# B&R Automation Studio project PT_KB_V01 (part 10)

#### Cyclic.st - Cyclic code
```iecst
PROGRAM _CYCLIC
	(* ======================================================================== *)
	(* 1) Komunikacioni, pogonski i AirRelease izvori                           *)
	(* ======================================================================== *)
	PT_Alarm.Comm.BRB2.Active := PGRad_Cmd.Aktivan AND NOT PGRad_BRB2Watchdog.Valid;
	PT_Alarm.Comm.IEBKB1.Active := PGRad_Cmd.Aktivan
		AND (PGRad.Ctrl.SelektovaniIzvor = _02_IEBKB1)
		AND (NOT PGRad_IEBKB1Prepared.CommValid OR NOT PGRad_IEBKB1Prepared.HeartbeatValid);
	PT_Alarm.Comm.BRB2RemoteFault.Active := PGRad_BRB2.BRB2Fault;
	PT_Alarm.Drive.PG_Pu01_VFD.Active := PG.Act.Pu._1.Alarm_FR;
	PT_Alarm.Drive.PG_Pu01_CAN.Active := PG.Act.Pu._1.Alarm_CAN;
	PT_Alarm.Drive.PG_Pu02_VFD.Active := PG.Act.Pu._2.Alarm_FR;
	PT_Alarm.Drive.PG_Pu02_CAN.Active := PG.Act.Pu._2.Alarm_CAN;
	PT_Alarm.AirRelease.PG_PV03.Active := PGRad_AirRelease.PV03.FB.AR_Output.AlarmActive;
	PT_Alarm.AirRelease.PG_PV04.Active := PGRad_AirRelease.PV04.FB.AR_Output.AlarmActive;

	PT_Alarm.Comm.BRB2.ResetAllowed := NOT PT_Alarm.Comm.BRB2.Active;
	PT_Alarm.Comm.IEBKB1.ResetAllowed := NOT PT_Alarm.Comm.IEBKB1.Active;
	PT_Alarm.Comm.BRB2RemoteFault.ResetAllowed := NOT PT_Alarm.Comm.BRB2RemoteFault.Active;
	PT_Alarm.Drive.PG_Pu01_VFD.ResetAllowed := NOT PT_Alarm.Drive.PG_Pu01_VFD.Active;
	PT_Alarm.Drive.PG_Pu01_CAN.ResetAllowed := NOT PT_Alarm.Drive.PG_Pu01_CAN.Active;
	PT_Alarm.Drive.PG_Pu02_VFD.ResetAllowed := NOT PT_Alarm.Drive.PG_Pu02_VFD.Active;
	PT_Alarm.Drive.PG_Pu02_CAN.ResetAllowed := NOT PT_Alarm.Drive.PG_Pu02_CAN.Active;
	PT_Alarm.AirRelease.PG_PV03.ResetAllowed := PGRad_AirRelease.PV03.FB.AR_Output.ResetAllowed;
	PT_Alarm.AirRelease.PG_PV04.ResetAllowed := PGRad_AirRelease.PV04.FB.AR_Output.ResetAllowed;
	PT_Alarm.AirRelease.PG_PV03.SourceCode := PGRad_AirRelease.PV03.FB.AR_Output.FaultCode;
	PT_Alarm.AirRelease.PG_PV04.SourceCode := PGRad_AirRelease.PV04.FB.AR_Output.FaultCode;

	(* ======================================================================== *)
	(* 2) IO_Modules: status, latch, potvrda i STOP svih fizickih modula       *)
	(* ======================================================================== *)
	PT_Alarm.IO.X20AI4622.Fault := NOT PT_Alarm.IO.X20AI4622.ModuleOk;
	PT_Alarm.IO.X20AI4622a.Fault := NOT PT_Alarm.IO.X20AI4622a.ModuleOk;
	PT_Alarm.IO.X20AI4622b.Fault := NOT PT_Alarm.IO.X20AI4622b.ModuleOk;
	PT_Alarm.IO.X20AI4622c.Fault := NOT PT_Alarm.IO.X20AI4622c.ModuleOk;
	PT_Alarm.IO.X20AI4622d.Fault := NOT PT_Alarm.IO.X20AI4622d.ModuleOk;
	PT_Alarm.IO.X20AO4622.Fault := NOT PT_Alarm.IO.X20AO4622.ModuleOk;
	PT_Alarm.IO.X20AO4622a.Fault := NOT PT_Alarm.IO.X20AO4622a.ModuleOk;
	PT_Alarm.IO.X20AO4622b.Fault := NOT PT_Alarm.IO.X20AO4622b.ModuleOk;
	PT_Alarm.IO.X20DI9371.Fault := NOT PT_Alarm.IO.X20DI9371.ModuleOk;
	PT_Alarm.IO.X20DI9371a.Fault := NOT PT_Alarm.IO.X20DI9371a.ModuleOk;
	PT_Alarm.IO.X20DI9371b.Fault := NOT PT_Alarm.IO.X20DI9371b.ModuleOk;
	PT_Alarm.IO.X20DO9322.Fault := NOT PT_Alarm.IO.X20DO9322.ModuleOk;
	PT_Alarm.IO.X20DO9322a.Fault := NOT PT_Alarm.IO.X20DO9322a.ModuleOk;
	PT_Alarm.IO.X20BC0083.Fault := NOT PT_Alarm.IO.X20BC0083.ModuleOk;
	PT_Alarm.IO.X20PS9400.Fault := NOT PT_Alarm.IO.X20PS9400.ModuleOk;
	PT_Alarm.IO.X20BT9100a.Fault := NOT PT_Alarm.IO.X20BT9100a.ModuleOk;
	PT_Alarm.IO.X67AI1323.Fault := NOT PT_Alarm.IO.X67AI1323.ModuleOk;
	PT_Alarm.IO.X67AI1333b.Fault := NOT PT_Alarm.IO.X67AI1333b.ModuleOk;
	PT_Alarm.IO.X67DI1371_L12.Fault := NOT PT_Alarm.IO.X67DI1371_L12.ModuleOk;
	PT_Alarm.IO.X67DM1321_L12.Fault := NOT PT_Alarm.IO.X67DM1321_L12.ModuleOk;
	PT_Alarm.IO.X20AI4622.Code := 41001; PT_Alarm.IO.X20AI4622.ResetAllowed := NOT PT_Alarm.IO.X20AI4622.Fault; PT_Alarm.IO.X20AI4622.Blocking := TRUE;
	PT_Alarm.IO.X20AI4622a.Code := 41002; PT_Alarm.IO.X20AI4622a.ResetAllowed := NOT PT_Alarm.IO.X20AI4622a.Fault; PT_Alarm.IO.X20AI4622a.Blocking := TRUE;
	PT_Alarm.IO.X20AI4622b.Code := 41003; PT_Alarm.IO.X20AI4622b.ResetAllowed := NOT PT_Alarm.IO.X20AI4622b.Fault; PT_Alarm.IO.X20AI4622b.Blocking := TRUE;
	PT_Alarm.IO.X20AI4622c.Code := 41004; PT_Alarm.IO.X20AI4622c.ResetAllowed := NOT PT_Alarm.IO.X20AI4622c.Fault; PT_Alarm.IO.X20AI4622c.Blocking := TRUE;
	PT_Alarm.IO.X20AI4622d.Code := 41005; PT_Alarm.IO.X20AI4622d.ResetAllowed := NOT PT_Alarm.IO.X20AI4622d.Fault; PT_Alarm.IO.X20AI4622d.Blocking := TRUE;
	PT_Alarm.IO.X20AO4622.Code := 41101; PT_Alarm.IO.X20AO4622.ResetAllowed := NOT PT_Alarm.IO.X20AO4622.Fault; PT_Alarm.IO.X20AO4622.Blocking := TRUE;
	PT_Alarm.IO.X20AO4622a.Code := 41102; PT_Alarm.IO.X20AO4622a.ResetAllowed := NOT PT_Alarm.IO.X20AO4622a.Fault; PT_Alarm.IO.X20AO4622a.Blocking := TRUE;
	PT_Alarm.IO.X20AO4622b.Code := 41103; PT_Alarm.IO.X20AO4622b.ResetAllowed := NOT PT_Alarm.IO.X20AO4622b.Fault; PT_Alarm.IO.X20AO4622b.Blocking := TRUE;
	PT_Alarm.IO.X20DI9371.Code := 41201; PT_Alarm.IO.X20DI9371.ResetAllowed := NOT PT_Alarm.IO.X20DI9371.Fault; PT_Alarm.IO.X20DI9371.Blocking := TRUE;
	PT_Alarm.IO.X20DI9371a.Code := 41202; PT_Alarm.IO.X20DI9371a.ResetAllowed := NOT PT_Alarm.IO.X20DI9371a.Fault; PT_Alarm.IO.X20DI9371a.Blocking := TRUE;
	PT_Alarm.IO.X20DI9371b.Code := 41203; PT_Alarm.IO.X20DI9371b.ResetAllowed := NOT PT_Alarm.IO.X20DI9371b.Fault; PT_Alarm.IO.X20DI9371b.Blocking := TRUE;
	PT_Alarm.IO.X20DO9322.Code := 41301; PT_Alarm.IO.X20DO9322.ResetAllowed := NOT PT_Alarm.IO.X20DO9322.Fault; PT_Alarm.IO.X20DO9322.Blocking := TRUE;
	PT_Alarm.IO.X20DO9322a.Code := 41302; PT_Alarm.IO.X20DO9322a.ResetAllowed := NOT PT_Alarm.IO.X20DO9322a.Fault; PT_Alarm.IO.X20DO9322a.Blocking := TRUE;
	PT_Alarm.IO.X20BC0083.Code := 41401; PT_Alarm.IO.X20BC0083.ResetAllowed := NOT PT_Alarm.IO.X20BC0083.Fault; PT_Alarm.IO.X20BC0083.Blocking := TRUE;
	PT_Alarm.IO.X20PS9400.Code := 41402; PT_Alarm.IO.X20PS9400.ResetAllowed := NOT PT_Alarm.IO.X20PS9400.Fault; PT_Alarm.IO.X20PS9400.Blocking := TRUE;
	PT_Alarm.IO.X20BT9100a.Code := 41403; PT_Alarm.IO.X20BT9100a.ResetAllowed := NOT PT_Alarm.IO.X20BT9100a.Fault; PT_Alarm.IO.X20BT9100a.Blocking := TRUE;
	PT_Alarm.IO.X67AI1323.Code := 41501; PT_Alarm.IO.X67AI1323.ResetAllowed := NOT PT_Alarm.IO.X67AI1323.Fault; PT_Alarm.IO.X67AI1323.Blocking := TRUE;
	PT_Alarm.IO.X67AI1333b.Code := 41502; PT_Alarm.IO.X67AI1333b.ResetAllowed := NOT PT_Alarm.IO.X67AI1333b.Fault; PT_Alarm.IO.X67AI1333b.Blocking := TRUE;
	PT_Alarm.IO.X67DI1371_L12.Code := 41601; PT_Alarm.IO.X67DI1371_L12.ResetAllowed := NOT PT_Alarm.IO.X67DI1371_L12.Fault; PT_Alarm.IO.X67DI1371_L12.Blocking := TRUE;
	PT_Alarm.IO.X67DM1321_L12.Code := 41701; PT_Alarm.IO.X67DM1321_L12.ResetAllowed := NOT PT_Alarm.IO.X67DM1321_L12.Fault; PT_Alarm.IO.X67DM1321_L12.Blocking := TRUE;
	IF PT_Alarm.IO.X20AI4622.Fault OR PT_Alarm.IO.X20AI4622a.Fault OR PT_Alarm.IO.X20AI4622b.Fault OR PT_Alarm.IO.X20AI4622c.Fault OR PT_Alarm.IO.X20AI4622d.Fault OR PT_Alarm.IO.X20AO4622.Fault OR PT_Alarm.IO.X20AO4622a.Fault OR PT_Alarm.IO.X20AO4622b.Fault OR PT_Alarm.IO.X20DI9371.Fault OR PT_Alarm.IO.X20DI9371a.Fault OR PT_Alarm.IO.X20DI9371b.Fault OR PT_Alarm.IO.X20DO9322.Fault OR PT_Alarm.IO.X20DO9322a.Fault OR PT_Alarm.IO.X20BC0083.Fault OR PT_Alarm.IO.X20PS9400.Fault OR PT_Alarm.IO.X20BT9100a.Fault OR PT_Alarm.IO.X67AI1323.Fault OR PT_Alarm.IO.X67AI1333b.Fault OR PT_Alarm.IO.X67DI1371_L12.Fault OR PT_Alarm.IO.X67DM1321_L12.Fault THEN
		PT_Alarm.IO.X20AI4622.Latched := PT_Alarm.IO.X20AI4622.Latched OR PT_Alarm.IO.X20AI4622.Fault;
		PT_Alarm.IO.X20AI4622a.Latched := PT_Alarm.IO.X20AI4622a.Latched OR PT_Alarm.IO.X20AI4622a.Fault;
		PT_Alarm.IO.X20AI4622b.Latched := PT_Alarm.IO.X20AI4622b.Latched OR PT_Alarm.IO.X20AI4622b.Fault;
		PT_Alarm.IO.X20AI4622c.Latched := PT_Alarm.IO.X20AI4622c.Latched OR PT_Alarm.IO.X20AI4622c.Fault;
		PT_Alarm.IO.X20AI4622d.Latched := PT_Alarm.IO.X20AI4622d.Latched OR PT_Alarm.IO.X20AI4622d.Fault;
		PT_Alarm.IO.X20AO4622.Latched := PT_Alarm.IO.X20AO4622.Latched OR PT_Alarm.IO.X20AO4622.Fault;
		PT_Alarm.IO.X20AO4622a.Latched := PT_Alarm.IO.X20AO4622a.Latched OR PT_Alarm.IO.X20AO4622a.Fault;
		PT_Alarm.IO.X20AO4622b.Latched := PT_Alarm.IO.X20AO4622b.Latched OR PT_Alarm.IO.X20AO4622b.Fault;
		PT_Alarm.IO.X20DI9371.Latched := PT_Alarm.IO.X20DI9371.Latched OR PT_Alarm.IO.X20DI9371.Fault;
		PT_Alarm.IO.X20DI9371a.Latched := PT_Alarm.IO.X20DI9371a.Latched OR PT_Alarm.IO.X20DI9371a.Fault;
		PT_Alarm.IO.X20DI9371b.Latched := PT_Alarm.IO.X20DI9371b.Latched OR PT_Alarm.IO.X20DI9371b.Fault;
		PT_Alarm.IO.X20DO9322.Latched := PT_Alarm.IO.X20DO9322.Latched OR PT_Alarm.IO.X20DO9322.Fault;
		PT_Alarm.IO.X20DO9322a.Latched := PT_Alarm.IO.X20DO9322a.Latched OR PT_Alarm.IO.X20DO9322a.Fault;
		PT_Alarm.IO.X20BC0083.Latched := PT_Alarm.IO.X20BC0083.Latched OR PT_Alarm.IO.X20BC0083.Fault;
		PT_Alarm.IO.X20PS9400.Latched := PT_Alarm.IO.X20PS9400.Latched OR PT_Alarm.IO.X20PS9400.Fault;
		PT_Alarm.IO.X20BT9100a.Latched := PT_Alarm.IO.X20BT9100a.Latched OR PT_Alarm.IO.X20BT9100a.Fault;
		PT_Alarm.IO.X67AI1323.Latched := PT_Alarm.IO.X67AI1323.Latched OR PT_Alarm.IO.X67AI1323.Fault;
		PT_Alarm.IO.X67AI1333b.Latched := PT_Alarm.IO.X67AI1333b.Latched OR PT_Alarm.IO.X67AI1333b.Fault;
		PT_Alarm.IO.X67DI1371_L12.Latched := PT_Alarm.IO.X67DI1371_L12.Latched OR PT_Alarm.IO.X67DI1371_L12.Fault;
		PT_Alarm.IO.X67DM1321_L12.Latched := PT_Alarm.IO.X67DM1321_L12.Latched OR PT_Alarm.IO.X67DM1321_L12.Fault;
	END_IF;
	IF PT_Alarm.Cmd.ResetAlarmRecords THEN
		IF PT_Alarm.IO.X20AI4622.ResetAllowed THEN PT_Alarm.IO.X20AI4622.Latched := FALSE; END_IF;
		IF PT_Alarm.IO.X20AI4622a.ResetAllowed THEN PT_Alarm.IO.X20AI4622a.Latched := FALSE; END_IF;
		IF PT_Alarm.IO.X20AI4622b.ResetAllowed THEN PT_Alarm.IO.X20AI4622b.Latched := FALSE; END_IF;
		IF PT_Alarm.IO.X20AI4622c.ResetAllowed THEN PT_Alarm.IO.X20AI4622c.Latched := FALSE; END_IF;
		IF PT_Alarm.IO.X20AI4622d.ResetAllowed THEN PT_Alarm.IO.X20AI4622d.Latched := FALSE; END_IF;
		IF PT_Alarm.IO.X20AO4622.ResetAllowed THEN PT_Alarm.IO.X20AO4622.Latched := FALSE; END_IF;
		IF PT_Alarm.IO.X20AO4622a.ResetAllowed THEN PT_Alarm.IO.X20AO4622a.Latched := FALSE; END_IF;
		IF PT_Alarm.IO.X20AO4622b.ResetAllowed THEN PT_Alarm.IO.X20AO4622b.Latched := FALSE; END_IF;
		IF PT_Alarm.IO.X20DI9371.ResetAllowed THEN PT_Alarm.IO.X20DI9371.Latched := FALSE; END_IF;
		IF PT_Alarm.IO.X20DI9371a.ResetAllowed THEN PT_Alarm.IO.X20DI9371a.Latched := FALSE; END_IF;
		IF PT_Alarm.IO.X20DI9371b.ResetAllowed THEN PT_Alarm.IO.X20DI9371b.Latched := FALSE; END_IF;
		IF PT_Alarm.IO.X20DO9322.ResetAllowed THEN PT_Alarm.IO.X20DO9322.Latched := FALSE; END_IF;
		IF PT_Alarm.IO.X20DO9322a.ResetAllowed THEN PT_Alarm.IO.X20DO9322a.Latched := FALSE; END_IF;
		IF PT_Alarm.IO.X20BC0083.ResetAllowed THEN PT_Alarm.IO.X20BC0083.Latched := FALSE; END_IF;
		IF PT_Alarm.IO.X20PS9400.ResetAllowed THEN PT_Alarm.IO.X20PS9400.Latched := FALSE; END_IF;
		IF PT_Alarm.IO.X20BT9100a.ResetAllowed THEN PT_Alarm.IO.X20BT9100a.Latched := FALSE; END_IF;
		IF PT_Alarm.IO.X67AI1323.ResetAllowed THEN PT_Alarm.IO.X67AI1323.Latched := FALSE; END_IF;
		IF PT_Alarm.IO.X67AI1333b.ResetAllowed THEN PT_Alarm.IO.X67AI1333b.Latched := FALSE; END_IF;
		IF PT_Alarm.IO.X67DI1371_L12.ResetAllowed THEN PT_Alarm.IO.X67DI1371_L12.Latched := FALSE; END_IF;
		IF PT_Alarm.IO.X67DM1321_L12.ResetAllowed THEN PT_Alarm.IO.X67DM1321_L12.Latched := FALSE; END_IF;
	END_IF;
	PT_Alarm.IO.AnyFault :=
		PT_Alarm.IO.X20AI4622.Fault OR PT_Alarm.IO.X20AI4622a.Fault OR PT_Alarm.IO.X20AI4622b.Fault OR
		PT_Alarm.IO.X20AI4622c.Fault OR PT_Alarm.IO.X20AI4622d.Fault OR PT_Alarm.IO.X20AO4622.Fault OR
		PT_Alarm.IO.X20AO4622a.Fault OR PT_Alarm.IO.X20AO4622b.Fault OR PT_Alarm.IO.X20DI9371.Fault OR
		PT_Alarm.IO.X20DI9371a.Fault OR PT_Alarm.IO.X20DI9371b.Fault OR PT_Alarm.IO.X20DO9322.Fault OR
		PT_Alarm.IO.X20DO9322a.Fault OR PT_Alarm.IO.X20BC0083.Fault OR PT_Alarm.IO.X20PS9400.Fault OR
		PT_Alarm.IO.X20BT9100a.Fault OR PT_Alarm.IO.X67AI1323.Fault OR PT_Alarm.IO.X67AI1333b.Fault OR
		PT_Alarm.IO.X67DI1371_L12.Fault OR PT_Alarm.IO.X67DM1321_L12.Fault;
	PT_Alarm.IO.AnyLatched :=
		PT_Alarm.IO.X20AI4622.Latched OR PT_Alarm.IO.X20AI4622a.Latched OR PT_Alarm.IO.X20AI4622b.Latched OR
		PT_Alarm.IO.X20AI4622c.Latched OR PT_Alarm.IO.X20AI4622d.Latched OR PT_Alarm.IO.X20AO4622.Latched OR
		PT_Alarm.IO.X20AO4622a.Latched OR PT_Alarm.IO.X20AO4622b.Latched OR PT_Alarm.IO.X20DI9371.Latched OR
		PT_Alarm.IO.X20DI9371a.Latched OR PT_Alarm.IO.X20DI9371b.Latched OR PT_Alarm.IO.X20DO9322.Latched OR
		PT_Alarm.IO.X20DO9322a.Latched OR PT_Alarm.IO.X20BC0083.Latched OR PT_Alarm.IO.X20PS9400.Latched OR
		PT_Alarm.IO.X20BT9100a.Latched OR PT_Alarm.IO.X67AI1323.Latched OR PT_Alarm.IO.X67AI1333b.Latched OR
		PT_Alarm.IO.X67DI1371_L12.Latched OR PT_Alarm.IO.X67DM1321_L12.Latched;
	PT_Alarm.IO.StopRequest := PT_Alarm.IO.AnyFault OR PT_Alarm.IO.AnyLatched;
	IF PT_Alarm.IO.FirstOutCode = 0 AND PT_Alarm.IO.AnyFault THEN
		IF PT_Alarm.IO.X20AI4622.Fault THEN PT_Alarm.IO.FirstOutCode := 41001;
		ELSIF PT_Alarm.IO.X20AI4622a.Fault THEN PT_Alarm.IO.FirstOutCode := 41002;
		ELSIF PT_Alarm.IO.X20AI4622b.Fault THEN PT_Alarm.IO.FirstOutCode := 41003;
		ELSIF PT_Alarm.IO.X20AI4622c.Fault THEN PT_Alarm.IO.FirstOutCode := 41004;
		ELSIF PT_Alarm.IO.X20AI4622d.Fault THEN PT_Alarm.IO.FirstOutCode := 41005;
		ELSIF PT_Alarm.IO.X20AO4622.Fault THEN PT_Alarm.IO.FirstOutCode := 41101;
		ELSIF PT_Alarm.IO.X20AO4622a.Fault THEN PT_Alarm.IO.FirstOutCode := 41102;
		ELSIF PT_Alarm.IO.X20AO4622b.Fault THEN PT_Alarm.IO.FirstOutCode := 41103;
		ELSIF PT_Alarm.IO.X20DI9371.Fault THEN PT_Alarm.IO.FirstOutCode := 41201;
		ELSIF PT_Alarm.IO.X20DI9371a.Fault THEN PT_Alarm.IO.FirstOutCode := 41202;
		ELSIF PT_Alarm.IO.X20DI9371b.Fault THEN PT_Alarm.IO.FirstOutCode := 41203;
		ELSIF PT_Alarm.IO.X20DO9322.Fault THEN PT_Alarm.IO.FirstOutCode := 41301;
		ELSIF PT_Alarm.IO.X20DO9322a.Fault THEN PT_Alarm.IO.FirstOutCode := 41302;
		ELSIF PT_Alarm.IO.X20BC0083.Fault THEN PT_Alarm.IO.FirstOutCode := 41401;
		ELSIF PT_Alarm.IO.X20PS9400.Fault THEN PT_Alarm.IO.FirstOutCode := 41402;
		ELSIF PT_Alarm.IO.X20BT9100a.Fault THEN PT_Alarm.IO.FirstOutCode := 41403;
		ELSIF PT_Alarm.IO.X67AI1323.Fault THEN PT_Alarm.IO.FirstOutCode := 41501;
		ELSIF PT_Alarm.IO.X67AI1333b.Fault THEN PT_Alarm.IO.FirstOutCode := 41502;
		ELSIF PT_Alarm.IO.X67DI1371_L12.Fault THEN PT_Alarm.IO.FirstOutCode := 41601;
		ELSIF PT_Alarm.IO.X67DM1321_L12.Fault THEN PT_Alarm.IO.FirstOutCode := 41701;
		END_IF;
	END_IF;

	(* ======================================================================== *)
	(* 3) Postojeci procesni FaultCode u imenovane alarmne zapise               *)
	(* ======================================================================== *)
	PT_Alarm.Process.ValveRequestConflict.Active := FALSE;
	PT_Alarm.Process.V01CloseTimeout.Active := FALSE;
	PT_Alarm.Process.V02OpenTimeout.Active := FALSE;
	PT_Alarm.Process.V02CloseTimeout.Active := FALSE;
	PT_Alarm.Process.V01OpenTimeout.Active := FALSE;
	PT_Alarm.Process.V01CloseIEBStopTimeout.Active := FALSE;
	PT_Alarm.Process.IEBFlowStopTimeout.Active := FALSE;
	PT_Alarm.Process.V05CloseTimeout.Active := FALSE;
	PT_Alarm.Process.IEBFlowStartTimeout.Active := FALSE;
	PT_Alarm.Process.BRB2FlowNotConfirmed.Active := FALSE;
	PT_Alarm.Process.BRB2TemperatureNotReached.Active := FALSE;
	PT_Alarm.Process.PT06HighPressure.Active := FALSE;
	PT_Alarm.Process.TransferIEBFlowNotZero.Active := FALSE;
	PT_Alarm.Process.TransferV05CloseTimeout.Active := FALSE;
	PT_Alarm.Process.TransferV01CloseTimeout.Active := FALSE;
	PT_Alarm.Process.TransferV02OpenTimeout.Active := FALSE;
	PT_Alarm.Process.TransferBRB2FlowNotConfirmed.Active := FALSE;

	IF PGRad_Status.Fault THEN
		CASE PGRad_Status.FaultCode OF
			10: PT_Alarm.Process.ValveRequestConflict.Active := TRUE;
			11: PT_Alarm.Process.V01CloseTimeout.Active := TRUE;
			12: PT_Alarm.Process.V02OpenTimeout.Active := TRUE;
			13: PT_Alarm.Process.V02CloseTimeout.Active := TRUE;
			14: PT_Alarm.Process.V01OpenTimeout.Active := TRUE;
			15: PT_Alarm.Process.V01CloseIEBStopTimeout.Active := TRUE;
			16: PT_Alarm.Process.IEBFlowStopTimeout.Active := TRUE;
			17: PT_Alarm.Process.V05CloseTimeout.Active := TRUE;
			18: PT_Alarm.Process.IEBFlowStartTimeout.Active := TRUE;
			21: PT_Alarm.Process.BRB2FlowNotConfirmed.Active := TRUE;
			22: PT_Alarm.Process.BRB2TemperatureNotReached.Active := TRUE;
			23: PT_Alarm.Process.PT06HighPressure.Active := TRUE;
			31: PT_Alarm.Process.TransferIEBFlowNotZero.Active := TRUE;
			32: PT_Alarm.Process.TransferV05CloseTimeout.Active := TRUE;
			33: PT_Alarm.Process.TransferV01CloseTimeout.Active := TRUE;
			34: PT_Alarm.Process.TransferV02OpenTimeout.Active := TRUE;
			35: PT_Alarm.Process.TransferBRB2FlowNotConfirmed.Active := TRUE;
		END_CASE;
	END_IF;

	PT_Alarm.Process.ValveRequestConflict.ResetAllowed := NOT PGRad_Status.Fault;
	PT_Alarm.Process.V01CloseTimeout.ResetAllowed := NOT PGRad_Status.Fault;
	PT_Alarm.Process.V02OpenTimeout.ResetAllowed := NOT PGRad_Status.Fault;
	PT_Alarm.Process.V02CloseTimeout.ResetAllowed := NOT PGRad_Status.Fault;
	PT_Alarm.Process.V01OpenTimeout.ResetAllowed := NOT PGRad_Status.Fault;
	PT_Alarm.Process.V01CloseIEBStopTimeout.ResetAllowed := NOT PGRad_Status.Fault;
	PT_Alarm.Process.IEBFlowStopTimeout.ResetAllowed := NOT PGRad_Status.Fault;
	PT_Alarm.Process.V05CloseTimeout.ResetAllowed := NOT PGRad_Status.Fault;
	PT_Alarm.Process.IEBFlowStartTimeout.ResetAllowed := NOT PGRad_Status.Fault;
	PT_Alarm.Process.BRB2FlowNotConfirmed.ResetAllowed := NOT PGRad_Status.Fault;
	PT_Alarm.Process.BRB2TemperatureNotReached.ResetAllowed := NOT PGRad_Status.Fault;
	PT_Alarm.Process.PT06HighPressure.ResetAllowed := NOT PGRad_Status.Fault;
	PT_Alarm.Process.TransferIEBFlowNotZero.ResetAllowed := NOT PGRad_Status.Fault;
	PT_Alarm.Process.TransferV05CloseTimeout.ResetAllowed := NOT PGRad_Status.Fault;
	PT_Alarm.Process.TransferV01CloseTimeout.ResetAllowed := NOT PGRad_Status.Fault;
	PT_Alarm.Process.TransferV02OpenTimeout.ResetAllowed := NOT PGRad_Status.Fault;
	PT_Alarm.Process.TransferBRB2FlowNotConfirmed.ResetAllowed := NOT PGRad_Status.Fault;

	(* ======================================================================== *)
	(* 3) Latch i first-out memorija                                            *)
	(* ======================================================================== *)
	IF PT_Alarm.Comm.BRB2.Active THEN
		PT_Alarm.Comm.BRB2.Latched := TRUE;
	END_IF;
	IF PT_Alarm.Comm.IEBKB1.Active THEN
		PT_Alarm.Comm.IEBKB1.Latched := TRUE;
	END_IF;
	IF PT_Alarm.Comm.BRB2RemoteFault.Active THEN
		PT_Alarm.Comm.BRB2RemoteFault.Latched := TRUE;
	END_IF;
	IF PT_Alarm.Drive.PG_Pu01_VFD.Active THEN
		PT_Alarm.Drive.PG_Pu01_VFD.Latched := TRUE;
	END_IF;
	IF PT_Alarm.Drive.PG_Pu01_CAN.Active THEN
		PT_Alarm.Drive.PG_Pu01_CAN.Latched := TRUE;
	END_IF;
	IF PT_Alarm.Drive.PG_Pu02_VFD.Active THEN
		PT_Alarm.Drive.PG_Pu02_VFD.Latched := TRUE;
	END_IF;
	IF PT_Alarm.Drive.PG_Pu02_CAN.Active THEN
		PT_Alarm.Drive.PG_Pu02_CAN.Latched := TRUE;
	END_IF;
	IF PGRad_AirRelease.PV03.FB.AR_Output.AlarmLatched THEN
		PT_Alarm.AirRelease.PG_PV03.Latched := TRUE;
	END_IF;
	IF PGRad_AirRelease.PV04.FB.AR_Output.AlarmLatched THEN
		PT_Alarm.AirRelease.PG_PV04.Latched := TRUE;
	END_IF;

	IF PT_Alarm.Process.ValveRequestConflict.Active THEN
		PT_Alarm.Process.ValveRequestConflict.Latched := TRUE;
	END_IF;
	IF PT_Alarm.Process.V01CloseTimeout.Active THEN
		PT_Alarm.Process.V01CloseTimeout.Latched := TRUE;
	END_IF;
	IF PT_Alarm.Process.V02OpenTimeout.Active THEN
		PT_Alarm.Process.V02OpenTimeout.Latched := TRUE;
	END_IF;
	IF PT_Alarm.Process.V02CloseTimeout.Active THEN
		PT_Alarm.Process.V02CloseTimeout.Latched := TRUE;
	END_IF;
	IF PT_Alarm.Process.V01OpenTimeout.Active THEN
		PT_Alarm.Process.V01OpenTimeout.Latched := TRUE;
	END_IF;
	IF PT_Alarm.Process.V01CloseIEBStopTimeout.Active THEN
		PT_Alarm.Process.V01CloseIEBStopTimeout.Latched := TRUE;
	END_IF;
	IF PT_Alarm.Process.IEBFlowStopTimeout.Active THEN
		PT_Alarm.Process.IEBFlowStopTimeout.Latched := TRUE;
	END_IF;
	IF PT_Alarm.Process.V05CloseTimeout.Active THEN
		PT_Alarm.Process.V05CloseTimeout.Latched := TRUE;
	END_IF;
	IF PT_Alarm.Process.IEBFlowStartTimeout.Active THEN
		PT_Alarm.Process.IEBFlowStartTimeout.Latched := TRUE;
	END_IF;
	IF PT_Alarm.Process.BRB2FlowNotConfirmed.Active THEN
		PT_Alarm.Process.BRB2FlowNotConfirmed.Latched := TRUE;
	END_IF;
	IF PT_Alarm.Process.BRB2TemperatureNotReached.Active THEN
		PT_Alarm.Process.BRB2TemperatureNotReached.Latched := TRUE;
	END_IF;
	IF PT_Alarm.Process.PT06HighPressure.Active THEN
		PT_Alarm.Process.PT06HighPressure.Latched := TRUE;
	END_IF;
	IF PT_Alarm.Process.TransferIEBFlowNotZero.Active THEN
		PT_Alarm.Process.TransferIEBFlowNotZero.Latched := TRUE;
	END_IF;
	IF PT_Alarm.Process.TransferV05CloseTimeout.Active THEN
		PT_Alarm.Process.TransferV05CloseTimeout.Latched := TRUE;
	END_IF;
	IF PT_Alarm.Process.TransferV01CloseTimeout.Active THEN
		PT_Alarm.Process.TransferV01CloseTimeout.Latched := TRUE;
	END_IF;
	IF PT_Alarm.Process.TransferV02OpenTimeout.Active THEN
		PT_Alarm.Process.TransferV02OpenTimeout.Latched := TRUE;
	END_IF;
	IF PT_Alarm.Process.TransferBRB2FlowNotConfirmed.Active THEN
		PT_Alarm.Process.TransferBRB2FlowNotConfirmed.Latched := TRUE;
	END_IF;

	IF PT_Alarm.Summary.FirstOutCode = 0 THEN
		IF PT_Alarm.Comm.BRB2.Active THEN
			PT_Alarm.Summary.FirstOutCode := PT_Alarm.Comm.BRB2.Code;
		ELSIF PT_Alarm.Comm.IEBKB1.Active THEN
			PT_Alarm.Summary.FirstOutCode := PT_Alarm.Comm.IEBKB1.Code;
		ELSIF PT_Alarm.Comm.BRB2RemoteFault.Active THEN
			PT_Alarm.Summary.FirstOutCode := PT_Alarm.Comm.BRB2RemoteFault.Code;
		ELSIF PT_Alarm.Drive.PG_Pu01_VFD.Active THEN
			PT_Alarm.Summary.FirstOutCode := PT_Alarm.Drive.PG_Pu01_VFD.Code;
		ELSIF PT_Alarm.Drive.PG_Pu01_CAN.Active THEN
			PT_Alarm.Summary.FirstOutCode := PT_Alarm.Drive.PG_Pu01_CAN.Code;
		ELSIF PT_Alarm.Drive.PG_Pu02_VFD.Active THEN
			PT_Alarm.Summary.FirstOutCode := PT_Alarm.Drive.PG_Pu02_VFD.Code;
		ELSIF PT_Alarm.Drive.PG_Pu02_CAN.Active THEN
			PT_Alarm.Summary.FirstOutCode := PT_Alarm.Drive.PG_Pu02_CAN.Code;
		ELSIF PGRad_Status.Fault THEN
			PT_Alarm.Summary.FirstOutCode := 25000 + USINT_TO_UINT(PGRad_Status.FaultCode);
		ELSIF PGRad_AirRelease.PV03.FB.AR_Output.AlarmLatched THEN
			PT_Alarm.Summary.FirstOutCode := PT_Alarm.AirRelease.PG_PV03.Code;
		ELSIF PGRad_AirRelease.PV04.FB.AR_Output.AlarmLatched THEN
			PT_Alarm.Summary.FirstOutCode := PT_Alarm.AirRelease.PG_PV04.Code;
		END_IF;
	END_IF;

	(* ======================================================================== *)
	(* 4) Operatorska potvrda i reset alarmnog zapisa                           *)
	(* ======================================================================== *)
	IF PT_Alarm.Cmd.AcknowledgeAll THEN
		PT_Alarm.Comm.BRB2.Acknowledged := PT_Alarm.Comm.BRB2.Latched;
		PT_Alarm.Comm.IEBKB1.Acknowledged := PT_Alarm.Comm.IEBKB1.Latched;
		PT_Alarm.Comm.BRB2RemoteFault.Acknowledged := PT_Alarm.Comm.BRB2RemoteFault.Latched;
		PT_Alarm.Drive.PG_Pu01_VFD.Acknowledged := PT_Alarm.Drive.PG_Pu01_VFD.Latched;
		PT_Alarm.Drive.PG_Pu01_CAN.Acknowledged := PT_Alarm.Drive.PG_Pu01_CAN.Latched;
		PT_Alarm.Drive.PG_Pu02_VFD.Acknowledged := PT_Alarm.Drive.PG_Pu02_VFD.Latched;
		PT_Alarm.Drive.PG_Pu02_CAN.Acknowledged := PT_Alarm.Drive.PG_Pu02_CAN.Latched;
		PT_Alarm.Process.ValveRequestConflict.Acknowledged := PT_Alarm.Process.ValveRequestConflict.Latched;
		PT_Alarm.Process.V01CloseTimeout.Acknowledged := PT_Alarm.Process.V01CloseTimeout.Latched;
		PT_Alarm.Process.V02OpenTimeout.Acknowledged := PT_Alarm.Process.V02OpenTimeout.Latched;
		PT_Alarm.Process.V02CloseTimeout.Acknowledged := PT_Alarm.Process.V02CloseTimeout.Latched;
		PT_Alarm.Process.V01OpenTimeout.Acknowledged := PT_Alarm.Process.V01OpenTimeout.Latched;
		PT_Alarm.Process.V01CloseIEBStopTimeout.Acknowledged := PT_Alarm.Process.V01CloseIEBStopTimeout.Latched;
		PT_Alarm.Process.IEBFlowStopTimeout.Acknowledged := PT_Alarm.Process.IEBFlowStopTimeout.Latched;
		PT_Alarm.Process.V05CloseTimeout.Acknowledged := PT_Alarm.Process.V05CloseTimeout.Latched;
		PT_Alarm.Process.IEBFlowStartTimeout.Acknowledged := PT_Alarm.Process.IEBFlowStartTimeout.Latched;
		PT_Alarm.Process.BRB2FlowNotConfirmed.Acknowledged := PT_Alarm.Process.BRB2FlowNotConfirmed.Latched;
		PT_Alarm.Process.BRB2TemperatureNotReached.Acknowledged := PT_Alarm.Process.BRB2TemperatureNotReached.Latched;
		PT_Alarm.Process.PT06HighPressure.Acknowledged := PT_Alarm.Process.PT06HighPressure.Latched;
		PT_Alarm.Process.TransferIEBFlowNotZero.Acknowledged := PT_Alarm.Process.TransferIEBFlowNotZero.Latched;
		PT_Alarm.Process.TransferV05CloseTimeout.Acknowledged := PT_Alarm.Process.TransferV05CloseTimeout.Latched;
		PT_Alarm.Process.TransferV01CloseTimeout.Acknowledged := PT_Alarm.Process.TransferV01CloseTimeout.Latched;
		PT_Alarm.Process.TransferV02OpenTimeout.Acknowledged := PT_Alarm.Process.TransferV02OpenTimeout.Latched;
		PT_Alarm.Process.TransferBRB2FlowNotConfirmed.Acknowledged := PT_Alarm.Process.TransferBRB2FlowNotConfirmed.Latched;
		PT_Alarm.AirRelease.PG_PV03.Acknowledged := PT_Alarm.AirRelease.PG_PV03.Latched;
		PT_Alarm.AirRelease.PG_PV04.Acknowledged := PT_Alarm.AirRelease.PG_PV04.Latched;
	END_IF;

	IF PT_Alarm.Cmd.ResetAlarmRecords THEN
		IF PT_Alarm.Comm.BRB2.ResetAllowed THEN
			PT_Alarm.Comm.BRB2.Latched := FALSE;
			PT_Alarm.Comm.BRB2.Acknowledged := FALSE;
		END_IF;
		IF PT_Alarm.Comm.IEBKB1.ResetAllowed THEN
			PT_Alarm.Comm.IEBKB1.Latched := FALSE;
			PT_Alarm.Comm.IEBKB1.Acknowledged := FALSE;
		END_IF;
		IF PT_Alarm.Comm.BRB2RemoteFault.ResetAllowed THEN
			PT_Alarm.Comm.BRB2RemoteFault.Latched := FALSE;
			PT_Alarm.Comm.BRB2RemoteFault.Acknowledged := FALSE;
		END_IF;
		IF PT_Alarm.Drive.PG_Pu01_VFD.ResetAllowed THEN
			PT_Alarm.Drive.PG_Pu01_VFD.Latched := FALSE;
			PT_Alarm.Drive.PG_Pu01_VFD.Acknowledged := FALSE;
		END_IF;
		IF PT_Alarm.Drive.PG_Pu01_CAN.ResetAllowed THEN
			PT_Alarm.Drive.PG_Pu01_CAN.Latched := FALSE;
			PT_Alarm.Drive.PG_Pu01_CAN.Acknowledged := FALSE;
		END_IF;
		IF PT_Alarm.Drive.PG_Pu02_VFD.ResetAllowed THEN
			PT_Alarm.Drive.PG_Pu02_VFD.Latched := FALSE;
			PT_Alarm.Drive.PG_Pu02_VFD.Acknowledged := FALSE;
		END_IF;
		IF PT_Alarm.Drive.PG_Pu02_CAN.ResetAllowed THEN
			PT_Alarm.Drive.PG_Pu02_CAN.Latched := FALSE;
			PT_Alarm.Drive.PG_Pu02_CAN.Acknowledged := FALSE;
		END_IF;
		IF NOT PGRad_Status.Fault THEN
			PT_Alarm.Process.ValveRequestConflict.Latched := FALSE;
			PT_Alarm.Process.ValveRequestConflict.Acknowledged := FALSE;
			PT_Alarm.Process.V01CloseTimeout.Latched := FALSE;
			PT_Alarm.Process.V01CloseTimeout.Acknowledged := FALSE;
			PT_Alarm.Process.V02OpenTimeout.Latched := FALSE;
			PT_Alarm.Process.V02OpenTimeout.Acknowledged := FALSE;
			PT_Alarm.Process.V02CloseTimeout.Latched := FALSE;
			PT_Alarm.Process.V02CloseTimeout.Acknowledged := FALSE;
			PT_Alarm.Process.V01OpenTimeout.Latched := FALSE;
			PT_Alarm.Process.V01OpenTimeout.Acknowledged := FALSE;
			PT_Alarm.Process.V01CloseIEBStopTimeout.Latched := FALSE;
			PT_Alarm.Process.V01CloseIEBStopTimeout.Acknowledged := FALSE;
			PT_Alarm.Process.IEBFlowStopTimeout.Latched := FALSE;
			PT_Alarm.Process.IEBFlowStopTimeout.Acknowledged := FALSE;
			PT_Alarm.Process.V05CloseTimeout.Latched := FALSE;
			PT_Alarm.Process.V05CloseTimeout.Acknowledged := FALSE;
			PT_Alarm.Process.IEBFlowStartTimeout.Latched := FALSE;
			PT_Alarm.Process.IEBFlowStartTimeout.Acknowledged := FALSE;
			PT_Alarm.Process.BRB2FlowNotConfirmed.Latched := FALSE;
			PT_Alarm.Process.BRB2FlowNotConfirmed.Acknowledged := FALSE;
			PT_Alarm.Process.BRB2TemperatureNotReached.Latched := FALSE;
			PT_Alarm.Process.BRB2TemperatureNotReached.Acknowledged := FALSE;
			PT_Alarm.Process.PT06HighPressure.Latched := FALSE;
			PT_Alarm.Process.PT06HighPressure.Acknowledged := FALSE;
			PT_Alarm.Process.TransferIEBFlowNotZero.Latched := FALSE;
			PT_Alarm.Process.TransferIEBFlowNotZero.Acknowledged := FALSE;
			PT_Alarm.Process.TransferV05CloseTimeout.Latched := FALSE;
			PT_Alarm.Process.TransferV05CloseTimeout.Acknowledged := FALSE;
			PT_Alarm.Process.TransferV01CloseTimeout.Latched := FALSE;
			PT_Alarm.Process.TransferV01CloseTimeout.Acknowledged := FALSE;
			PT_Alarm.Process.TransferV02OpenTimeout.Latched := FALSE;
			PT_Alarm.Process.TransferV02OpenTimeout.Acknowledged := FALSE;
			PT_Alarm.Process.TransferBRB2FlowNotConfirmed.Latched := FALSE;
			PT_Alarm.Process.TransferBRB2FlowNotConfirmed.Acknowledged := FALSE;
		END_IF;
		IF PT_Alarm.AirRelease.PG_PV03.ResetAllowed THEN
			PT_Alarm.AirRelease.PG_PV03.Latched := FALSE;
			PT_Alarm.AirRelease.PG_PV03.Acknowledged := FALSE;
		END_IF;
		IF PT_Alarm.AirRelease.PG_PV04.ResetAllowed THEN
			PT_Alarm.AirRelease.PG_PV04.Latched := FALSE;
			PT_Alarm.AirRelease.PG_PV04.Acknowledged := FALSE;
		END_IF;
	END_IF;

	(* ======================================================================== *)
	(* 5) Zbirni status                                                         *)
	(* ======================================================================== *)
	ProcessAnyLatched := PT_Alarm.Process.ValveRequestConflict.Latched
		OR PT_Alarm.Process.V01CloseTimeout.Latched
		OR PT_Alarm.Process.V02OpenTimeout.Latched
		OR PT_Alarm.Process.V02CloseTimeout.Latched
		OR PT_Alarm.Process.V01OpenTimeout.Latched
		OR PT_Alarm.Process.V01CloseIEBStopTimeout.Latched
		OR PT_Alarm.Process.IEBFlowStopTimeout.Latched
		OR PT_Alarm.Process.V05CloseTimeout.Latched
		OR PT_Alarm.Process.IEBFlowStartTimeout.Latched
		OR PT_Alarm.Process.BRB2FlowNotConfirmed.Latched
		OR PT_Alarm.Process.BRB2TemperatureNotReached.Latched
		OR PT_Alarm.Process.PT06HighPressure.Latched
		OR PT_Alarm.Process.TransferIEBFlowNotZero.Latched
		OR PT_Alarm.Process.TransferV05CloseTimeout.Latched
		OR PT_Alarm.Process.TransferV01CloseTimeout.Latched
		OR PT_Alarm.Process.TransferV02OpenTimeout.Latched
		OR PT_Alarm.Process.TransferBRB2FlowNotConfirmed.Latched;
	ProcessAnyUnacknowledged :=
		(PT_Alarm.Process.ValveRequestConflict.Latched AND NOT PT_Alarm.Process.ValveRequestConflict.Acknowledged)
		OR (PT_Alarm.Process.V01CloseTimeout.Latched AND NOT PT_Alarm.Process.V01CloseTimeout.Acknowledged)
		OR (PT_Alarm.Process.V02OpenTimeout.Latched AND NOT PT_Alarm.Process.V02OpenTimeout.Acknowledged)
		OR (PT_Alarm.Process.V02CloseTimeout.Latched AND NOT PT_Alarm.Process.V02CloseTimeout.Acknowledged)
		OR (PT_Alarm.Process.V01OpenTimeout.Latched AND NOT PT_Alarm.Process.V01OpenTimeout.Acknowledged)
		OR (PT_Alarm.Process.V01CloseIEBStopTimeout.Latched AND NOT PT_Alarm.Process.V01CloseIEBStopTimeout.Acknowledged)
		OR (PT_Alarm.Process.IEBFlowStopTimeout.Latched AND NOT PT_Alarm.Process.IEBFlowStopTimeout.Acknowledged)
		OR (PT_Alarm.Process.V05CloseTimeout.Latched AND NOT PT_Alarm.Process.V05CloseTimeout.Acknowledged)
		OR (PT_Alarm.Process.IEBFlowStartTimeout.Latched AND NOT PT_Alarm.Process.IEBFlowStartTimeout.Acknowledged)
		OR (PT_Alarm.Process.BRB2FlowNotConfirmed.Latched AND NOT PT_Alarm.Process.BRB2FlowNotConfirmed.Acknowledged)
		OR (PT_Alarm.Process.BRB2TemperatureNotReached.Latched AND NOT PT_Alarm.Process.BRB2TemperatureNotReached.Acknowledged)
		OR (PT_Alarm.Process.PT06HighPressure.Latched AND NOT PT_Alarm.Process.PT06HighPressure.Acknowledged)
		OR (PT_Alarm.Process.TransferIEBFlowNotZero.Latched AND NOT PT_Alarm.Process.TransferIEBFlowNotZero.Acknowledged)
		OR (PT_Alarm.Process.TransferV05CloseTimeout.Latched AND NOT PT_Alarm.Process.TransferV05CloseTimeout.Acknowledged)
		OR (PT_Alarm.Process.TransferV01CloseTimeout.Latched AND NOT PT_Alarm.Process.TransferV01CloseTimeout.Acknowledged)
		OR (PT_Alarm.Process.TransferV02OpenTimeout.Latched AND NOT PT_Alarm.Process.TransferV02OpenTimeout.Acknowledged)
		OR (PT_Alarm.Process.TransferBRB2FlowNotConfirmed.Latched AND NOT PT_Alarm.Process.TransferBRB2FlowNotConfirmed.Acknowledged);

	PT_Alarm.Summary.ActiveCount := 0;
	PT_Alarm.Summary.LatchedCount := 0;
	IF PT_Alarm.Comm.BRB2.Active THEN
		PT_Alarm.Summary.ActiveCount := PT_Alarm.Summary.ActiveCount + 1;
	END_IF;
	IF PT_Alarm.Comm.IEBKB1.Active THEN
		PT_Alarm.Summary.ActiveCount := PT_Alarm.Summary.ActiveCount + 1;
	END_IF;
	IF PT_Alarm.Comm.BRB2RemoteFault.Active THEN
		PT_Alarm.Summary.ActiveCount := PT_Alarm.Summary.ActiveCount + 1;
	END_IF;
	IF PT_Alarm.Drive.PG_Pu01_VFD.Active THEN
		PT_Alarm.Summary.ActiveCount := PT_Alarm.Summary.ActiveCount + 1;
	END_IF;
	IF PT_Alarm.Drive.PG_Pu01_CAN.Active THEN
		PT_Alarm.Summary.ActiveCount := PT_Alarm.Summary.ActiveCount + 1;
	END_IF;
	IF PT_Alarm.Drive.PG_Pu02_VFD.Active THEN
		PT_Alarm.Summary.ActiveCount := PT_Alarm.Summary.ActiveCount + 1;
	END_IF;
	IF PT_Alarm.Drive.PG_Pu02_CAN.Active THEN
		PT_Alarm.Summary.ActiveCount := PT_Alarm.Summary.ActiveCount + 1;
	END_IF;
	IF PGRad_Status.Fault THEN
		PT_Alarm.Summary.ActiveCount := PT_Alarm.Summary.ActiveCount + 1;
	END_IF;
	IF PT_Alarm.AirRelease.PG_PV03.Active THEN
		PT_Alarm.Summary.ActiveCount := PT_Alarm.Summary.ActiveCount + 1;
	END_IF;
	IF PT_Alarm.AirRelease.PG_PV04.Active THEN
		PT_Alarm.Summary.ActiveCount := PT_Alarm.Summary.ActiveCount + 1;
	END_IF;

	IF PT_Alarm.Comm.BRB2.Latched THEN
		PT_Alarm.Summary.LatchedCount := PT_Alarm.Summary.LatchedCount + 1;
	END_IF;
	IF PT_Alarm.Comm.IEBKB1.Latched THEN
		PT_Alarm.Summary.LatchedCount := PT_Alarm.Summary.LatchedCount + 1;
	END_IF;
	IF PT_Alarm.Comm.BRB2RemoteFault.Latched THEN
		PT_Alarm.Summary.LatchedCount := PT_Alarm.Summary.LatchedCount + 1;
	END_IF;
	IF PT_Alarm.Drive.PG_Pu01_VFD.Latched THEN
		PT_Alarm.Summary.LatchedCount := PT_Alarm.Summary.LatchedCount + 1;
	END_IF;
	IF PT_Alarm.Drive.PG_Pu01_CAN.Latched THEN
		PT_Alarm.Summary.LatchedCount := PT_Alarm.Summary.LatchedCount + 1;
	END_IF;
	IF PT_Alarm.Drive.PG_Pu02_VFD.Latched THEN
		PT_Alarm.Summary.LatchedCount := PT_Alarm.Summary.LatchedCount + 1;
	END_IF;
	IF PT_Alarm.Drive.PG_Pu02_CAN.Latched THEN
		PT_Alarm.Summary.LatchedCount := PT_Alarm.Summary.LatchedCount + 1;
	END_IF;
	IF ProcessAnyLatched THEN
		PT_Alarm.Summary.LatchedCount := PT_Alarm.Summary.LatchedCount + 1;
	END_IF;
	IF PT_Alarm.AirRelease.PG_PV03.Latched THEN
		PT_Alarm.Summary.LatchedCount := PT_Alarm.Summary.LatchedCount + 1;
	END_IF;
	IF PT_Alarm.AirRelease.PG_PV04.Latched THEN
		PT_Alarm.Summary.LatchedCount := PT_Alarm.Summary.LatchedCount + 1;
	END_IF;

	PT_Alarm.Summary.AnyActive := (PT_Alarm.Summary.ActiveCount > 0) OR PT_Alarm.IO.AnyFault;
	PT_Alarm.Summary.AnyLatched := (PT_Alarm.Summary.LatchedCount > 0) OR PT_Alarm.IO.AnyLatched;
	PT_Alarm.Summary.AnyUnacknowledged :=
		(PT_Alarm.Comm.BRB2.Latched AND NOT PT_Alarm.Comm.BRB2.Acknowledged)
		OR (PT_Alarm.Comm.IEBKB1.Latched AND NOT PT_Alarm.Comm.IEBKB1.Acknowledged)
		OR (PT_Alarm.Comm.BRB2RemoteFault.Latched AND NOT PT_Alarm.Comm.BRB2RemoteFault.Acknowledged)
		OR (PT_Alarm.Drive.PG_Pu01_VFD.Latched AND NOT PT_Alarm.Drive.PG_Pu01_VFD.Acknowledged)
		OR (PT_Alarm.Drive.PG_Pu01_CAN.Latched AND NOT PT_Alarm.Drive.PG_Pu01_CAN.Acknowledged)
		OR (PT_Alarm.Drive.PG_Pu02_VFD.Latched AND NOT PT_Alarm.Drive.PG_Pu02_VFD.Acknowledged)
		OR (PT_Alarm.Drive.PG_Pu02_CAN.Latched AND NOT PT_Alarm.Drive.PG_Pu02_CAN.Acknowledged)
		OR ProcessAnyUnacknowledged
		OR (PT_Alarm.AirRelease.PG_PV03.Latched AND NOT PT_Alarm.AirRelease.PG_PV03.Acknowledged)
		OR (PT_Alarm.AirRelease.PG_PV04.Latched AND NOT PT_Alarm.AirRelease.PG_PV04.Acknowledged)
		OR PT_Alarm.IO.AnyLatched;
	PT_Alarm.Summary.AnyTrip := PT_Alarm.Comm.BRB2.Latched
		OR PT_Alarm.Comm.IEBKB1.Latched
		OR PT_Alarm.Comm.BRB2RemoteFault.Latched
		OR PT_Alarm.Drive.PG_Pu01_VFD.Latched
		OR PT_Alarm.Drive.PG_Pu01_CAN.Latched
		OR PT_Alarm.Drive.PG_Pu02_VFD.Latched
		OR PT_Alarm.Drive.PG_Pu02_CAN.Latched
		OR ProcessAnyLatched
		OR PT_Alarm.IO.StopRequest;
	PT_Alarm.Summary.RestartBlocked := PT_Alarm.Summary.AnyTrip OR PT_Alarm.IO.StopRequest;
	IF PT_Alarm.Summary.AnyTrip THEN
		PT_Alarm.Summary.HighestSeverity := 4;
	ELSIF PT_Alarm.Summary.AnyLatched THEN
		PT_Alarm.Summary.HighestSeverity := 3;
	ELSE
		PT_Alarm.Summary.HighestSeverity := 0;
	END_IF;
	IF NOT PT_Alarm.Summary.AnyLatched THEN
		PT_Alarm.Summary.FirstOutCode := 0;
	END_IF;
	IF NOT PT_Alarm.IO.AnyLatched THEN
		PT_Alarm.IO.FirstOutCode := 0;
	END_IF;
	IF PT_Alarm.Summary.FirstOutCode = 0 THEN
		PT_Alarm.Summary.FirstOutCode := PT_Alarm.IO.FirstOutCode;
	END_IF;

	(* ======================================================================== *)
	(* 7) Jednociklusne komande                                                  *)
	(* ======================================================================== *)
	PT_Alarm.ResetPulse.Devices := PT_Alarm.Cmd.ResetDevices;
	PT_Alarm.ResetPulse.Process := PT_Alarm.Cmd.ResetProcess;
	PT_Alarm.Cmd.AcknowledgeAll := FALSE;
	PT_Alarm.Cmd.ResetAlarmRecords := FALSE;
	PT_Alarm.Cmd.ResetDevices := FALSE;
	PT_Alarm.Cmd.ResetProcess := FALSE;
END_PROGRAM
```

#### Exit.st - Exit code
```iecst
PROGRAM _EXIT
	(* AlarmMgr nema resurse koji zahtevaju zatvaranje pri izlasku taska. *)
END_PROGRAM
```

#### Variables.var - Local variables
```iecst
VAR
	ProcessAnyLatched : BOOL; (* Najmanje jedan imenovani procesni alarm je memorisan. *)
	ProcessAnyUnacknowledged : BOOL; (* Najmanje jedan procesni alarm ceka potvrdu. *)
END_VAR
```

### Program Logical/Project/ValveResetSvc (IEC)

#### Cyclic.st - Cyclic code
```iecst
PROGRAM _CYCLIC
	(* ======================================================================== *)
	(* VALVE RESET SERVICE - RESET POJEDINACNIH I SVIH VENTILA                 *)
	(* ResetAlarm je impuls; posle validnog reseta Enable se obara jedan scan  *)
	(* i zatim ponovo podize, kako zahtevaju FB_V_EMV i FB_V_ON_OFF_FB.        *)
	(* ======================================================================== *)
	ResetPulse_01 := FALSE;
	ResetPulse_02 := FALSE;
	ResetPulse_03 := FALSE;
	ResetPulse_04 := FALSE;
	ResetPulse_05 := FALSE;
	ResetPulse_06 := FALSE;
	ResetPulse_07 := FALSE;

	ResetAllInProgress := ResetInProgress_01 OR ResetInProgress_02 OR ResetInProgress_03
		OR ResetInProgress_04 OR ResetInProgress_05 OR ResetInProgress_06 OR ResetInProgress_07;
	ResetAllDone := ResetDone_01 AND ResetDone_02 AND ResetDone_03 AND ResetDone_04
		AND ResetDone_05 AND ResetDone_06 AND ResetDone_07;
	ResetAllFault := ResetFault_01 OR ResetFault_02 OR ResetFault_03 OR ResetFault_04
		OR ResetFault_05 OR ResetFault_06 OR ResetFault_07;
	StateComment_01 := PG.Act.AV._1.V_Output.State_comment;
	FaultText_01 := PG.Act.AV._1.V_Output.FaultText;
	Diag_01 := PG.Act.AV._1.V_Output.Diag;
	StateComment_02 := PG.Act.AV._2.V_Output.State_comment;
	FaultText_02 := PG.Act.AV._2.V_Output.FaultText;
	Diag_02 := PG.Act.AV._2.V_Output.Diag;
	StateComment_03 := PG.Act.AV._3.V_Output.State_comment;
	FaultText_03 := PG.Act.AV._3.V_Output.FaultText;
	Diag_03 := PG.Act.AV._3.V_Output.Diag;
	StateComment_04 := PG.Act.AV._4.V_Output.State_comment;
	FaultText_04 := PG.Act.AV._4.V_Output.FaultText;
	Diag_04 := PG.Act.AV._4.V_Output.Diag;
	StateComment_05 := PG.Act.AV._5.V_Output.State_comment;
	FaultText_05 := PG.Act.AV._5.V_Output.FaultText;
	Diag_05 := PG.Act.AV._5.V_Output.Diag;
	StateComment_06 := PG.Act.AV._6.V_Output.State_comment;
	FaultText_06 := PG.Act.AV._6.V_Output.FaultText;
	Diag_06 := PG.Act.AV._6.V_Output.Diag;
	StateComment_07 := PG.Act.AV._7.V_Output.State_comment;
	FaultText_07 := PG.Act.AV._7.V_Output.FaultText;
	Diag_07 := PG.Act.AV._7.V_Output.Diag;
	ValveAlarmActive := PG.Act.AV._1.V_Output.FaultLatched
		OR PG.Act.AV._2.V_Output.FaultLatched
		OR PG.Act.AV._3.V_Output.FaultLatched
		OR PG.Act.AV._4.V_Output.FaultLatched
		OR PG.Act.AV._5.V_Output.FaultLatched
		OR PG.Act.AV._6.V_Output.FaultLatched
		OR PG.Act.AV._7.V_Output.FaultLatched;

//	PG.Act.AV._1.V_Input.Enable := NOT Disable_01;
	PG.Act.AV._1.V_Input.ResetAlarm := ResetPulse_01;
	IF (Reset_01 OR ResetAll) AND NOT PrevReset_01 AND NOT ResetInProgress_01 THEN
		ResetDone_01 := FALSE;
		ResetFault_01 := NOT PG.Act.AV._1.V_Output.ResetAllowed;
		IF PG.Act.AV._1.V_Output.ResetAllowed THEN ResetPulse_01 := TRUE; ResetInProgress_01 := TRUE; END_IF;
	END_IF;
	IF ResetInProgress_01 THEN
		IF ResetPulse_01 THEN ResetPulse_01 := FALSE; Disable_01 := TRUE;
		ELSIF Disable_01 THEN Disable_01 := FALSE; ResetInProgress_01 := FALSE; ResetDone_01 := TRUE; END_IF;
	END_IF;
	IF PG.Act.AV._1.V_Output.FaultLatched THEN ResetDone_01 := FALSE; END_IF;

	PG.Act.AV._2.V_Input.Enable := NOT Disable_02;
	PG.Act.AV._2.V_Input.ResetAlarm := ResetPulse_02;
	IF (Reset_02 OR ResetAll) AND NOT PrevReset_02 AND NOT ResetInProgress_02 THEN
		ResetDone_02 := FALSE;
		ResetFault_02 := NOT PG.Act.AV._2.V_Output.ResetAllowed;
		IF PG.Act.AV._2.V_Output.ResetAllowed THEN ResetPulse_02 := TRUE; ResetInProgress_02 := TRUE; END_IF;
	END_IF;
	IF ResetInProgress_02 THEN
		IF ResetPulse_02 THEN ResetPulse_02 := FALSE; Disable_02 := TRUE;
		ELSIF Disable_02 THEN Disable_02 := FALSE; ResetInProgress_02 := FALSE; ResetDone_02 := TRUE; END_IF;
	END_IF;
	IF PG.Act.AV._2.V_Output.FaultLatched THEN ResetDone_02 := FALSE; END_IF;

	PG.Act.AV._3.V_Input.Enable := NOT Disable_03;
	PG.Act.AV._3.V_Input.ResetAlarm := ResetPulse_03;
	IF (Reset_03 OR ResetAll) AND NOT PrevReset_03 AND NOT ResetInProgress_03 THEN
		ResetDone_03 := FALSE;
		ResetFault_03 := NOT PG.Act.AV._3.V_Output.ResetAllowed;
		IF PG.Act.AV._3.V_Output.ResetAllowed THEN ResetPulse_03 := TRUE; ResetInProgress_03 := TRUE; END_IF;
	END_IF;
	IF ResetInProgress_03 THEN
		IF ResetPulse_03 THEN ResetPulse_03 := FALSE; Disable_03 := TRUE;
		ELSIF Disable_03 THEN Disable_03 := FALSE; ResetInProgress_03 := FALSE; ResetDone_03 := TRUE; END_IF;
	END_IF;
	IF PG.Act.AV._3.V_Output.FaultLatched THEN ResetDone_03 := FALSE; END_IF;

	PG.Act.AV._4.V_Input.Enable := NOT Disable_04;
	PG.Act.AV._4.V_Input.ResetAlarm := ResetPulse_04;
	IF (Reset_04 OR ResetAll) AND NOT PrevReset_04 AND NOT ResetInProgress_04 THEN
		ResetDone_04 := FALSE;
		ResetFault_04 := NOT PG.Act.AV._4.V_Output.ResetAllowed;
		IF PG.Act.AV._4.V_Output.ResetAllowed THEN ResetPulse_04 := TRUE; ResetInProgress_04 := TRUE; END_IF;
	END_IF;
	IF ResetInProgress_04 THEN
		IF ResetPulse_04 THEN ResetPulse_04 := FALSE; Disable_04 := TRUE;
		ELSIF Disable_04 THEN Disable_04 := FALSE; ResetInProgress_04 := FALSE; ResetDone_04 := TRUE; END_IF;
	END_IF;
	IF PG.Act.AV._4.V_Output.FaultLatched THEN ResetDone_04 := FALSE; END_IF;

	PG.Act.AV._5.V_Input.Enable := NOT Disable_05;
	PG.Act.AV._5.V_Input.ResetAlarm := ResetPulse_05;
	IF (Reset_05 OR ResetAll) AND NOT PrevReset_05 AND NOT ResetInProgress_05 THEN
		ResetDone_05 := FALSE;
		ResetFault_05 := NOT PG.Act.AV._5.V_Output.ResetAllowed;
		IF PG.Act.AV._5.V_Output.ResetAllowed THEN ResetPulse_05 := TRUE; ResetInProgress_05 := TRUE; END_IF;
	END_IF;
	IF ResetInProgress_05 THEN
		IF ResetPulse_05 THEN ResetPulse_05 := FALSE; Disable_05 := TRUE;
		ELSIF Disable_05 THEN Disable_05 := FALSE; ResetInProgress_05 := FALSE; ResetDone_05 := TRUE; END_IF;
	END_IF;
	IF PG.Act.AV._5.V_Output.FaultLatched THEN ResetDone_05 := FALSE; END_IF;

	PG.Act.AV._6.V_Input.Enable := NOT Disable_06;
	PG.Act.AV._6.V_Input.ResetAlarm := ResetPulse_06;
	IF (Reset_06 OR ResetAll) AND NOT PrevReset_06 AND NOT ResetInProgress_06 THEN
		ResetDone_06 := FALSE;
		ResetFault_06 := NOT PG.Act.AV._6.V_Output.ResetAllowed;
		IF PG.Act.AV._6.V_Output.ResetAllowed THEN ResetPulse_06 := TRUE; ResetInProgress_06 := TRUE; END_IF;
	END_IF;
	IF ResetInProgress_06 THEN
		IF ResetPulse_06 THEN ResetPulse_06 := FALSE; Disable_06 := TRUE;
		ELSIF Disable_06 THEN Disable_06 := FALSE; ResetInProgress_06 := FALSE; ResetDone_06 := TRUE; END_IF;
	END_IF;
	IF PG.Act.AV._6.V_Output.FaultLatched THEN ResetDone_06 := FALSE; END_IF;

	PG.Act.AV._7.V_Input.Enable := NOT Disable_07;
	PG.Act.AV._7.V_Input.ResetAlarm := ResetPulse_07;
	IF (Reset_07 OR ResetAll) AND NOT PrevReset_07 AND NOT ResetInProgress_07 THEN
		ResetDone_07 := FALSE;
		ResetFault_07 := NOT PG.Act.AV._7.V_Output.ResetAllowed;
		IF PG.Act.AV._7.V_Output.ResetAllowed THEN ResetPulse_07 := TRUE; ResetInProgress_07 := TRUE; END_IF;
	END_IF;
	IF ResetInProgress_07 THEN
		IF ResetPulse_07 THEN ResetPulse_07 := FALSE; Disable_07 := TRUE;
		ELSIF Disable_07 THEN Disable_07 := FALSE; ResetInProgress_07 := FALSE; ResetDone_07 := TRUE; END_IF;
	END_IF;
	IF PG.Act.AV._7.V_Output.FaultLatched THEN ResetDone_07 := FALSE; END_IF;

	PrevResetAll := ResetAll;
	PrevReset_01 := Reset_01;
	PrevReset_02 := Reset_02;
	PrevReset_03 := Reset_03;
	PrevReset_04 := Reset_04;
	PrevReset_05 := Reset_05;
	PrevReset_06 := Reset_06;
	PrevReset_07 := Reset_07;
END_PROGRAM
```

#### Variables.var - Local variables
```iecst
VAR
	ResetAll : BOOL; (* HMI zahtev za reset svih ventila. *)
	Reset_01 : BOOL; (* HMI zahtev za reset PG_V01. *)
	Reset_02 : BOOL; (* HMI zahtev za reset PG_V02. *)
	Reset_03 : BOOL; (* HMI zahtev za reset PG_V03. *)
	Reset_04 : BOOL; (* HMI zahtev za reset PG_V04. *)
	Reset_05 : BOOL; (* HMI zahtev za reset PG_V05. *)
	Reset_06 : BOOL; (* HMI zahtev za reset PG_V06. *)
	Reset_07 : BOOL; (* HMI zahtev za reset PG_V07. *)
	ResetInProgress_01 : BOOL;
	ResetInProgress_02 : BOOL;
	ResetInProgress_03 : BOOL;
	ResetInProgress_04 : BOOL;
	ResetInProgress_05 : BOOL;
	ResetInProgress_06 : BOOL;
	ResetInProgress_07 : BOOL;
	ResetDone_01 : BOOL;
	ResetDone_02 : BOOL;
	ResetDone_03 : BOOL;
	ResetDone_04 : BOOL;
	ResetDone_05 : BOOL;
	ResetDone_06 : BOOL;
	ResetDone_07 : BOOL;
	ResetFault_01 : BOOL;
	ResetFault_02 : BOOL;
	ResetFault_03 : BOOL;
	ResetFault_04 : BOOL;
	ResetFault_05 : BOOL;
	ResetFault_06 : BOOL;
	ResetFault_07 : BOOL;
	ResetAllInProgress : BOOL;
	ResetAllDone : BOOL;
	ResetAllFault : BOOL;
	PrevResetAll : BOOL;
	PrevReset_01 : BOOL;
	PrevReset_02 : BOOL;
	PrevReset_03 : BOOL;
	PrevReset_04 : BOOL;
	PrevReset_05 : BOOL;
	PrevReset_06 : BOOL;
	PrevReset_07 : BOOL;
	ResetPulse_01 : BOOL;
	ResetPulse_02 : BOOL;
	ResetPulse_03 : BOOL;
	ResetPulse_04 : BOOL;
	ResetPulse_05 : BOOL;
	ResetPulse_06 : BOOL;
	ResetPulse_07 : BOOL;
	Disable_01 : BOOL;
	Disable_02 : BOOL;
	Disable_03 : BOOL;
	Disable_04 : BOOL;
	Disable_05 : BOOL;
	Disable_06 : BOOL;
	Disable_07 : BOOL;
	StateComment_01 : STRING[80];
	FaultText_01 : STRING[80];
	Diag_01 : STRING[80];
	StateComment_02 : STRING[80];
	FaultText_02 : STRING[80];
	Diag_02 : STRING[80];
	StateComment_03 : STRING[80];
	FaultText_03 : STRING[80];
	Diag_03 : STRING[80];
	StateComment_04 : STRING[80];
	FaultText_04 : STRING[80];
	Diag_04 : STRING[80];
	StateComment_05 : STRING[80];
	FaultText_05 : STRING[80];
	Diag_05 : STRING[80];
	StateComment_06 : STRING[80];
	FaultText_06 : STRING[80];
	Diag_06 : STRING[80];
	StateComment_07 : STRING[80];
	FaultText_07 : STRING[80];
	Diag_07 : STRING[80];
	ValveAlarmActive : BOOL; (* Zbirni alarm bilo kog PG_V01..PG_V07 ventila. *)
END_VAR
```

#### Init.st
```iecst
PROGRAM _INIT
	ResetAll := FALSE;
	Reset_01 := FALSE;
	Reset_02 := FALSE;
	Reset_03 := FALSE;
	Reset_04 := FALSE;
	Reset_05 := FALSE;
	Reset_06 := FALSE;
	Reset_07 := FALSE;
END_PROGRAM
```

#### Exit.st
```iecst
PROGRAM _EXIT
END_PROGRAM
```

Listed in the project but not available here: Logical/Libraries/BR_Lib/Constants.var, Logical/Libraries/NashCan1/Constants.var, Logical/DeviceCtrl/Init.st, Logical/DeviceCtrl/Cyclic.st, Logical/HMI_Svc/Exit.st, Logical/HMI_Svc/Variables.var, Logical/CAN/Init.st, Logical/CAN/Exit.st, Logical/Config2_ATV/Cyclic.st, Logical/Config2_ATV/Exit.st, Logical/Project/DeviceCtrl/Exit.st, Logical/Project/HMI_Svc/Exit.st
